TYPE ST_PostRunReport :
STRUCT
	runNo				: INT;
	analyst				: STRING(100);
	comment				: STRING(100);
	softwareVersion		: STRING(100);
	sysMasterRevision	: STRING(100);
	sysSettingsRevision	: STRING(100);
	meterVelocity		: STRING(100);
	runVelocity			: STRING(100);
	emptyTubesFactor	: STRING(100);
	fillTubesFactor		: STRING(100);
	solvent1NameRevision: STRING(100);
	solvent2NameRevision: STRING(100);
	solvent3NameRevision: STRING(100);
	solvent4NameRevision: STRING(100);
	timeEventStarted	: STRING(100);
	timeEventCompleted	: STRING(100);
	methodID			: INT;
	CalibrationNo		: INT;
END_STRUCT
END_TYPE

(* stored: Version 1.1.0.1, ProductVersion 3.1.4024.15
   DUT ST_PostRunReport: Id {f2068320-89cd-429f-819a-3a8eabf602d9} *)
